TYPE ST_PNOutput_ParallelOperation :
STRUCT
	statusbits		:	DWORD;
	ActivePower		:	DWORD;
	ReactivePower	:	DWORD;
END_STRUCT
END_TYPE

(* stored: Version 1.1.0.1, ProductVersion 3.1.4024.12
   DUT ST_PNOutput_ParallelOperation: Id {b22b8f93-2968-42a3-85ad-534a2e1643ee} *)
